% RSLogix 500 project Part_Counter_with_Analog_Safety_Override.RSS, saved by version 8.30.00.16 %
PROJECT "UNTITLED"    % processor: Bul.1763 MicroLogix 1100 Series B %

PROGRAM FILES
  LAD 2 "MAIN"  5 rungs
  LAD 3 "DIGITAL IO"  5 rungs
  LAD 4 "ANALOG IO"  2 rungs

DATA FILES
  O0 OUTPUT  7 elements
  I1 INPUT  13 elements
  S2 STATUS  66 elements
  B3 BINARY  1 elements
  T4 TIMER  1 elements
  C5 COUNTER  1 elements
  R6 CONTROL  1 elements
  N7 INTEGER  1 elements
  F8 FLOAT  1 elements

LADDER 2 "MAIN"
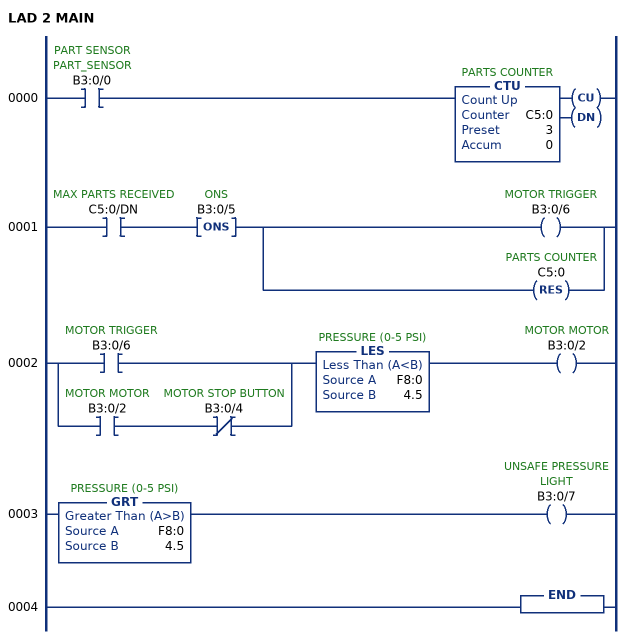
% Rung: 0 %
SOR XIC B3:0/0 CTU C5:0 3 0 EOR
%   B3:0/0  PART_SENSOR  "PART SENSOR" %
%   C5:0  "PARTS COUNTER" %
% Rung: 1 %
SOR XIC C5:0/DN ONS B3:0/5 BST OTE B3:0/6 NXB RES C5:0 BND EOR
%   C5:0/DN  "MAX PARTS RECEIVED" %
%   B3:0/5  "ONS" %
%   B3:0/6  "MOTOR TRIGGER" %
%   C5:0  "PARTS COUNTER" %
% Rung: 2 %
SOR BST XIC B3:0/6 NXB XIC B3:0/2 XIO B3:0/4 BND LES F8:0 4.5 OTE B3:0/2 EOR
%   B3:0/6  "MOTOR TRIGGER" %
%   B3:0/2  MOTOR  "MOTOR" %
%   B3:0/4  "MOTOR STOP BUTTON" %
%   F8:0  "PRESSURE (0-5 PSI)" %
% Rung: 3 %
SOR GRT F8:0 4.5 OTE B3:0/7 EOR
%   F8:0  "PRESSURE (0-5 PSI)" %
%   B3:0/7  "UNSAFE PRESSURE LIGHT" %
% Rung: 4 %
SOR END EOR

LADDER 3 "DIGITAL IO"
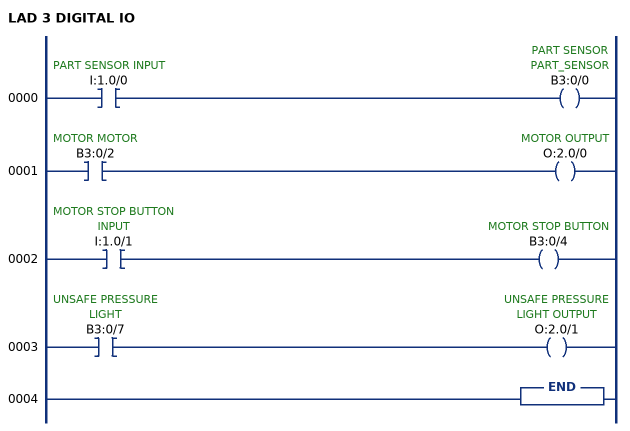
% Rung: 0 %
SOR XIC I:1.0/0 OTE B3:0/0 EOR
%   I:1.0/0  "PART SENSOR INPUT" %
%   B3:0/0  PART_SENSOR  "PART SENSOR" %
% Rung: 1 %
SOR XIC B3:0/2 OTE O:2.0/0 EOR
%   B3:0/2  MOTOR  "MOTOR" %
%   O:2.0/0  "MOTOR OUTPUT" %
% Rung: 2 %
SOR XIC I:1.0/1 OTE B3:0/4 EOR
%   I:1.0/1  "MOTOR STOP BUTTON INPUT" %
%   B3:0/4  "MOTOR STOP BUTTON" %
% Rung: 3 %
SOR XIC B3:0/7 OTE O:2.0/1 EOR
%   B3:0/7  "UNSAFE PRESSURE LIGHT" %
%   O:2.0/1  "UNSAFE PRESSURE LIGHT OUTPUT" %
% Rung: 4 %
SOR END EOR

LADDER 4 "ANALOG IO"
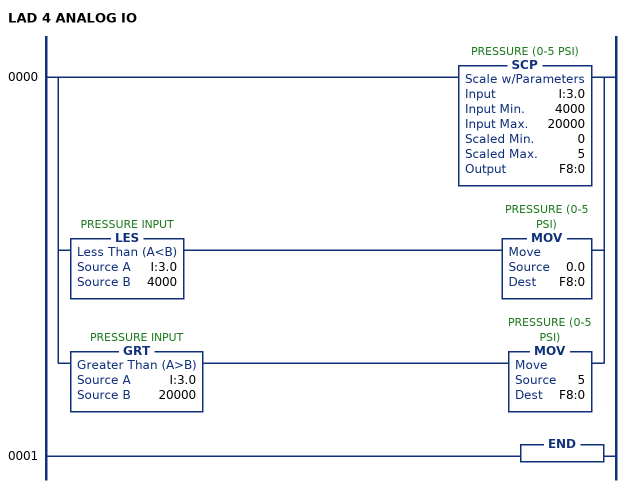
% Rung: 0 %
SOR BST SCP I:3.0 4000 20000 0 5 F8:0 NXB LES I:3.0 4000 MOV 0.0 F8:0 NXB GRT I:3.0 20000 MOV 5 F8:0 BND EOR
%   I:3.0  "PRESSURE INPUT" %
%   F8:0  "PRESSURE (0-5 PSI)" %
% Rung: 1 %
SOR END EOR

OTHER DOCUMENTED ADDRESSES
  B3:0/3  "STOP BUTTON"

DATA TABLE (non-zero values as saved)
DATA C5
% .PRE .ACC %
% C5:0 % 3 0
